// TIA Portal project "analog" (V14)

(* hardware
DEVICE "HMI_1"  KTP400 Basic PN
   slot 0: "KTP400 Basic PN"  KTP400 Basic PN  6AV2 123-2DB03-0AX0  14.0.1.0
   slot 1: "HMI_RT_1"  KTP400 Basic PN  6AV2 123-2DB03-0AX0  14.0.1.0
   slot 5: "HMI_1.IE_CP_1"  PROFINET Interface  14.0.1.0
      slot 1: "PROFINET Interface_1"  PROFINET Interface
         slot 1: "Port_1"  Port
DEVICE "S7-1200 station_1"  S7-1200 Station
   slot 0: "Rack_0"  S7-1200 Rack  Rack  V1.0
   slot 1: "PLC_1"  CPU 1212C DC/DC/DC  6ES7 212-1AE40-0XB0  V4.2
*)

// ===== PLC "PLC_1"  CPU 1212C DC/DC/DC =====

VAR_GLOBAL   // PLC tag table "Default tag table"
   "start" AT %I0.0 : Bool;
   "stop" AT %I0.1 : Bool;
   "bien tam" AT %M0.0 : Bool;
   "Tag_1" AT %IW64 : Word;
   "gia tri" AT %MD2 : DWord;
   "nhietdo" AT %MD6 : Real;
   "Tag_2" AT %Q0.0 : Bool;
   "Tag_3" AT %Q0.1 : Bool;
   "Tag_4" AT %Q0.2 : Bool;
   "start_hmi" AT %M0.1 : Bool;
   "stop_hmi" AT %M0.2 : Bool;
END_VAR

ORGANIZATION_BLOCK "Main"   // OB1, LAD, ProgramCycle
TITLE = "Main Program Sweep (Cycle)"
{ S7_Optimized_Access := 'TRUE' }
VERSION : 0.1
   VAR_INPUT
      Initial_Call : Bool;   // Initial call of this OB
      Remanence : Bool;   // =True, if remanent data are available
   END_VAR
BEGIN

REGION Network 1
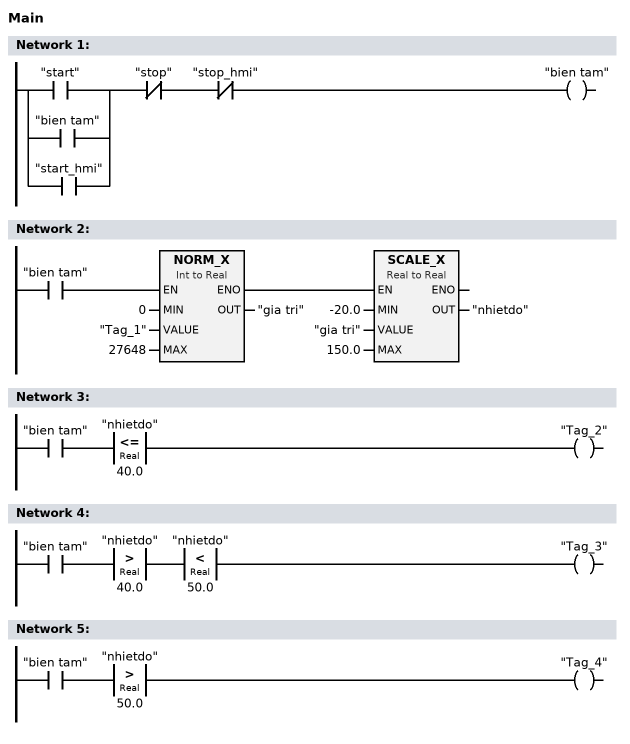
   RUNG wire#powerrail
      Contact( "start" )
      wire#w1
      I_Contact( "stop" )
      I_Contact( "stop_hmi" )
      Coil( "bien tam" )
   END_RUNG
   RUNG wire#powerrail
      Contact( "bien tam" )
   END_RUNG wire#w1
   RUNG wire#powerrail
      Contact( "start_hmi" )
   END_RUNG wire#w1
   // the same network as SCL:
   "bien tam" := ("start" OR "bien tam" OR "start_hmi") AND NOT "stop" AND NOT "stop_hmi";
END_REGION

REGION Network 2
   RUNG wire#powerrail
      Contact( "bien tam" )
      { S7_Templates := "[SrcType := Int, DestType := Real]" } Normalize(min := 0, value := "Tag_1", max := 27648, out => "gia tri")
      { S7_Templates := "[SrcType := Real, DestType := Real]" } Scale(min := -20.0, value := "gia tri", max := 150.0, out => "nhietdo")
   END_RUNG
   // the same network as SCL:
   IF "bien tam" THEN
       "gia tri" := NORM_X(MIN := 0, VALUE := "Tag_1", MAX := 27648);
       "nhietdo" := SCALE_X(MIN := -20.0, VALUE := "gia tri", MAX := 150.0);
   END_IF;
END_REGION

REGION Network 3
   RUNG wire#powerrail
      Contact( "bien tam" )
      { S7_Templates := "SrcType := Real" } LE_Contact(in1 := "nhietdo", in2 := 40.0)
      Coil( "Tag_2" )
   END_RUNG
   // the same network as SCL:
   "Tag_2" := "bien tam" AND ("nhietdo" <= 40.0);
END_REGION

REGION Network 4
   RUNG wire#powerrail
      Contact( "bien tam" )
      { S7_Templates := "SrcType := Real" } GT_Contact(in1 := "nhietdo", in2 := 40.0)
      { S7_Templates := "SrcType := Real" } LT_Contact(in1 := "nhietdo", in2 := 50.0)
      Coil( "Tag_3" )
   END_RUNG
   // the same network as SCL:
   "Tag_3" := "bien tam" AND ("nhietdo" > 40.0) AND ("nhietdo" < 50.0);
END_REGION

REGION Network 5
   RUNG wire#powerrail
      Contact( "bien tam" )
      { S7_Templates := "SrcType := Real" } GT_Contact(in1 := "nhietdo", in2 := 50.0)
      Coil( "Tag_4" )
   END_RUNG
   // the same network as SCL:
   "Tag_4" := "bien tam" AND ("nhietdo" > 50.0);
END_REGION
END_ORGANIZATION_BLOCK

(* ===== HMI "HMI_RT_1" =====
system functions are stored by id; their names below are inferred from use
connection "HMI_Connection_1": ETHERNET, SMART_S7_1200_OMS

HMI tags "Default tag table"
   "start" : Bool = PLC start AT %I0.0, 100 ms
   "stop" : Bool = PLC stop AT %I0.1, 100 ms
   "start_hmi" : Bool = PLC start_hmi AT %M0.1, 100 ms
   "bien tam" : Bool = PLC "bien tam" AT %M0.0, 100 ms
   "stop_hmi" : Bool = PLC stop_hmi AT %M0.2, 100 ms
   "nhietdo" : Real = PLC nhietdo AT %MD6, 100 ms

Template "Template_1" 480x272
   Button "Exit" at 388,227 size 63x44; TextOff 'Exit'; PictureOff "ExitRuntime_KTP400_Basic_PN_TR"; PictureOn "ExitRuntime_KTP400_Basic_PN_TR"
      on Release: StopRuntime(0)
   Button "Template_Button" at 268,227 size 63x44; TextOff 'Text'
   Button "Template_Button_1" at 148,227 size 63x44; TextOff 'Text'
   Button "Start screen" at 28,227 size 63x44; TextOff 'Start screen'; PictureOff "NavigateHome_KTP400_Basic_PN_TR"; PictureOn "NavigateHome_KTP400_Basic_PN_TR"
      on Release: ActivateScreen("Root screen", 0)

screen "Root screen" 480x272, template "Template_1"
   TextField "HmiScreenItemData" at 47,12 size 384x22; Text 'Using analog to calculate temp'
   Button "Button_1" at 13,120 size 96x32; TextOff 'start'
      on Press: SetBit("start_hmi")
      on Release: ResetBit("start_hmi")
      Appearance <- "bien tam"
   Button "Button_2" at 160,120 size 96x32; TextOff 'stop'
      on Press: SetBit("stop_hmi")
      on Release: ResetBit("stop_hmi")
      Appearance <- "bien tam"
   IOField "I/O field_1" at 328,120 size 96x32; FormatPattern s999999999.999
      ProcessValue <- "nhietdo"
*)